TYPE TcoSmartFunctionKitResults :
STRUCT	
	Id: UINT;
	
END_STRUCT
END_TYPE

(* stored: Version 1.1.0.1
   DUT TcoSmartFunctionKitResults: Id {0ebb6877-3cce-41e1-861d-57af02882eb1} *)
